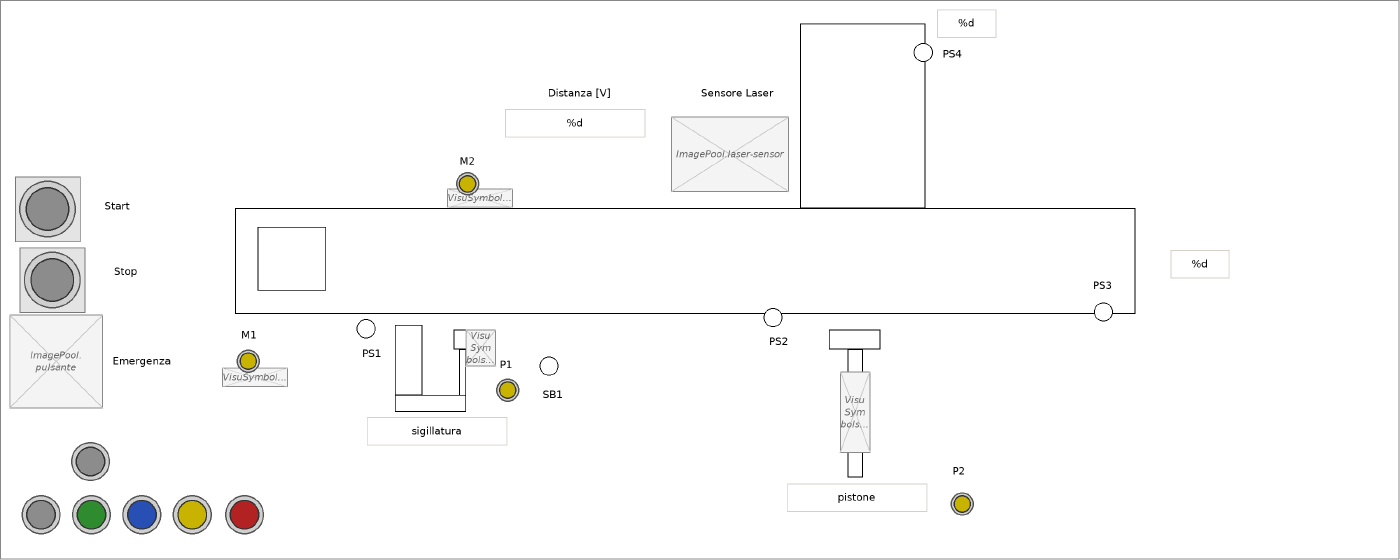
VISUALIZATION Visualization  // 1500x600
    RoundedRectangle (252,223 964x113)
    PushSwitch (16,189 70x70), variable: GVL.PB1, behaviour: TAP, style: Switch-PushSwitch-Gray
    Label (98,206 55x30), "Start"
    PushSwitch (21,265 70x70), variable: GVL.PB2, behaviour: TAP, style: Switch-PushSwitch-Gray
    Label (102,276 65x30), "Stop"
    Label (107,372 90x30), "Emergenza"
    Lamp1 (20,527 48x49), variable: GVL.L1, style: Lamp-Lamp1-Gray
    Lamp1 (74,527 48x49), variable: GVL.L2, style: Lamp-Lamp1-Green
    Lamp1 (128,527 48x49), variable: GVL.L3, style: Lamp-Lamp1-Blue
    Lamp1 (182,527 48x49), variable: GVL.L4, style: Lamp-Lamp1-Yellow
    Lamp1 (238,527 48x49), variable: GVL.L5, style: Lamp-Lamp1-Red
    Image (10,337 100x100), image: ImagePool.pulsante
        OnMouseClick: toggle GVL.PBE
    Textfield (843,518 150x30), "pistone"
    Rectangle (314,-68 198x134), angle 270
    RoundedRectangle (888,353 55x21)
    Rectangle (908,374 16x137)
    Image (900,398 32x87), image: VisuSymbols.Symbols.DoubleArrow4
    Rectangle (276,243 73x68)
    RoundedRectangle (486,353 19x21)
    Rectangle (492,374 7x51)
    Rectangle (423,423 76x18)
    Rectangle (423,348 29x75)
    Image (499,353 32x39), image: VisuSymbols.Symbols.DoubleArrow4
    Textfield (393,447 150x30), "sigillatura"
    Image (479,202 70x20), image: VisuSymbols.Symbols.ArrowBoldRight
    Image (238,394 70x20), image: VisuSymbols.Symbols.ArrowBoldRight
    Label (225,344 84x30), "M1"
    Label (459,158 84x30), "M2"
    Lamp1 (252,372 28x30), variable: GVL.M1, style: Lamp-Lamp1-Yellow
    Lamp1 (487,182 28x30), variable: GVL.M2, style: Lamp-Lamp1-Yellow
    Image (719,125 126x80), image: ImagePool.laser-sensor
    Lamp1 (1017,525 28x30), variable: GVL.P2, style: Lamp-Lamp1-Yellow
    Label (815,360 39x12), "PS2"
    Ellipse (818,330 20x20), colour toggle: GVL.PS2
        tap GVL.PS2
    Label (529,376 27x30), "P1"
    Lamp1 (530,403 28x30), variable: GVL.P1, style: Lamp-Lamp1-Yellow
    Ellipse (1172,324 20x20), colour toggle: GVL.PS3
        tap GVL.PS3
    Label (1162,300 39x12), "PS3"
    Textfield (1254,268 63x30), "%d", text variable: MAIN.CTU_BASSI.CV
    Lamp1 (73,470 48x49), variable: MAIN.STOP_RICHIESTO, style: Lamp-Lamp1-Gray
    Label (573,417 39x12), "SB1"
    Ellipse (578,382 20x20), colour toggle: GVL.SB1
        tap GVL.SB1
    Label (1014,490 27x30), "P2"
    Label (741,94 98x12), "Sensore Laser"
    Label (379,373 39x12), "PS1"
    Ellipse (382,342 20x20), colour toggle: GVL.PS1
        tap GVL.PS1
    Ellipse (979,46 20x20), colour toggle: GVL.PS4
        tap GVL.PS4
    Label (1001,52 39x12), "PS4"
    Textfield (1004,10 63x30), "%d", text variable: MAIN.CTU_ALTI.CV
    Textfield (541,117 150x30), "%d", text variable: GVL.LS1
        OnMouseClick: write the text variable via VisuDialogs.Numpad, min 0, max 10
    Label (572,94 98x12), "Distanza [V]"
END_VISUALIZATION

(* stored: Version 1.1.0.1, ProductVersion 3.1.4024.12
   Visu Visualization: Id {e3399594-b7fd-4589-9a49-3967da9e8e84} *)
